// TIA Portal V20 export
TYPE "typeCmHmiInterfaceSoftCam"
// stored: Access Published, Namespace Unit1.Em13
   STRUCT
      jrUnIoadingPnPAxisX : "Unit1.Em13.typeCmHmiInterfaceSoftCamjrUnIoadingPnPAxisX";
      jrUnIoadingPnPAxisZ : "Unit1.Em13.typeCmHmiInterfaceSoftCamjrUnIoadingPnPAxisZ";
      jrUnIoadingPnPAxisC : "Unit1.Em13.typeCmHmiInterfaceSoftCamjrUnIoadingPnPAxisC";
   END_STRUCT;
END_TYPE
